// Mitsubishi GX Works2 project: test_step motor   PLC: FX3U/FX3UC

PROGRAM MAIN
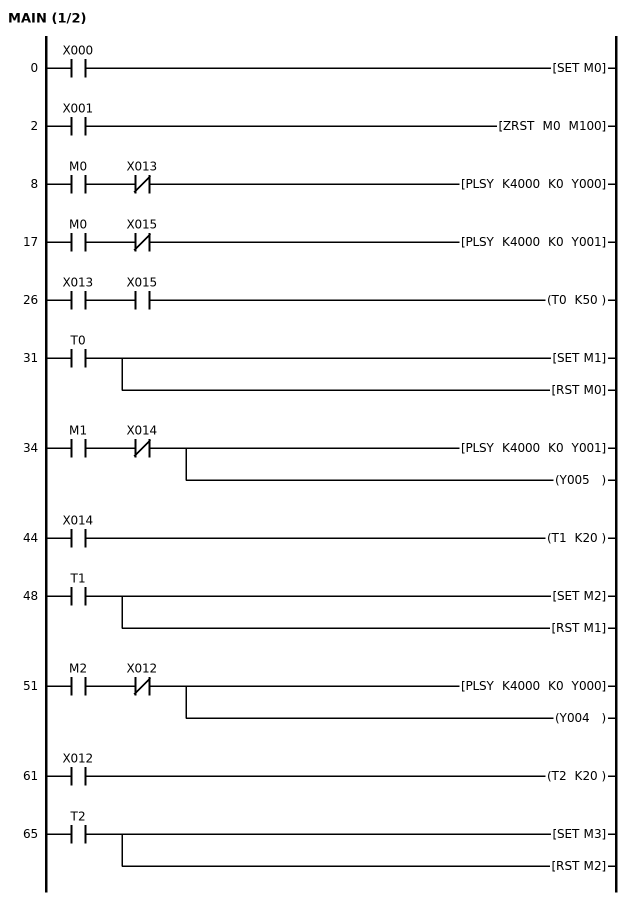
0     LD      X000
      SET     M0
2     LD      X001
      ZRST    M0 M100
8     LD      M0
      ANI     X013
      PLSY    K4000 K0 Y000
17    LD      M0
      ANI     X015
      PLSY    K4000 K0 Y001
26    LD      X013
      AND     X015
      OUT     T0 K50
31    LD      T0
      SET     M1
      RST     M0
34    LD      M1
      ANI     X014
      PLSY    K4000 K0 Y001
      OUT     Y005
44    LD      X014
      OUT     T1 K20
48    LD      T1
      SET     M2
      RST     M1
51    LD      M2
      ANI     X012
      PLSY    K4000 K0 Y000
      OUT     Y004
61    LD      X012
      OUT     T2 K20
65    LD      T2
      SET     M3
      RST     M2
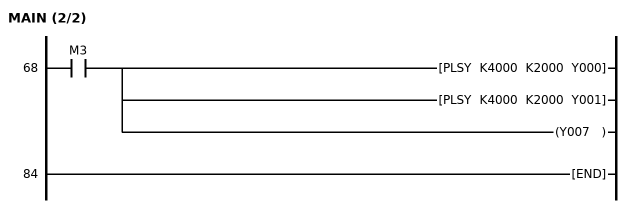
68    LD      M3
      PLSY    K4000 K2000 Y000
      PLSY    K4000 K2000 Y001
      OUT     Y007
84    END
END_PROGRAM
